Fanuc KAREL source: kd00019.KL

-- PROVISIONAL review KL for V1013-1; original PC SHA256 804466caa90b0d055bcb9e6a3d03cee5a3dfcce5b54d4b926520bb2fa476350c
-- Incomplete behavior may be omitted. Consult companion uncertainty JSON. Do not deploy.
PROGRAM KD00019
%NOLOCKGROUP
VAR
  I : INTEGER
  J : INTEGER
  B : BOOLEAN
  R : REAL
  S : STRING[80]
-- UNRESOLVED_DECL REC type=001100
BEGIN
  -- UNRESOLVED_PC offsets 5-16; opcodes 9D,22,32,35
  -- UNRESOLVED_PC offsets 26-48; opcodes 22,32,34,9D,52,22,32,35
  -- UNRESOLVED_PC offsets 58-62; opcodes 7F
END KD00019
